(* Logix 5000 project; controller Savage_Saw vendor 1 type 14 code 154 rev 37.11; software revision 37.01 *)

TASK MainTask (continuous, watchdog 500 ms) : Init, Inputs, MainProgram, Outputs

MODULES
   Local : vendor 1 type 14 code 154 (PointIO 0, rev 37.11)
      RMC : vendor 590 type 43 code 5 (Ethernet 192.168.3.12, rev 1.1, StandardDataDriven RPI 20 ms, StandardDataDriven RPI 20 ms)
      RemoteHPU : 1734-AENTR (Ethernet 192.168.3.11, rev 7.13, Output RPI 20 ms)
         AnalogIn5_6 : 1734-IE2V (PointIO 1, rev 3.4, Input RPI 80 ms)
         InputDC0_8 : 1734-IB8 (PointIO 2, rev 3.22)
         InputDC9_15 : 1734-IB8 (PointIO 3, rev 3.22)
         OutputDC4_7 : vendor 1 type 7 code 134 (PointIO 5, rev 3.2)
         OutputDC0_3 : vendor 1 type 7 code 134 (PointIO 4, rev 3.2)
      Analog4_5 : 1734-IE2V (PointIO 4, rev 3.1, Input RPI 80 ms)
      Analog0_1 : 1734-IE2V (PointIO 2, rev 3.5, Input RPI 80 ms)
      Analog2_3 : 1734-IE2V (PointIO 3, rev 3.4, Input RPI 80 ms)
      Discrete_IO : Embedded (PointIO 1, rev 37.11, Output RPI 20 ms)
      SpindleSpeed : 1734-OE2V (PointIO 5, rev 3.5, Output RPI 50 ms)
      Swarf_Outputs : 1734-OA4 (PointIO 7, rev 3.22, Output RPI 20 ms)
      Light_Outputs : 1734-OA4 (PointIO 8, rev 3.22, Output RPI 20 ms)
      HPU_Outputs : 1734-OA4 (PointIO 6, rev 3.22, Output RPI 20 ms)
END_MODULES

TYPE AxisData :
STRUCT
   PositionActual : REAL;
   FinalOutput : REAL;
   VelocityActual : REAL;
   PositionTarget : REAL;
   VelocityTarget : REAL;
   InPosition : BOOL;
   AtVelocity : BOOL;
   OpenLoop : BOOL;
   FaultInput : BOOL;
   LimitPos : BOOL;
   LimitNeg : BOOL;
   Stopped : BOOL;
   InputEstimated : BOOL;
   OutputEnabled : BOOL;
   TargetGeneratorDone : BOOL;
   TargetGeneratorStateA : BOOL;
   TargetGeneratorStateB : BOOL;
   DirectOutput : BOOL;
   Enabled : BOOL;
   ExternalHalt : BOOL;
   Halted : BOOL;
   ForceControlled : BOOL;
   ForceLimitEnabled : BOOL;
   ForceLimited : BOOL;
   AtForce : BOOL;
   ForceInputEstimated : BOOL;
   ForceTargetGeneratorDone : BOOL;
   ForceTargetGeneratorStateA : BOOL;
   ForceTargetGeneratorStateB : BOOL;
   TargetGeneratorBusy : BOOL;
   ForceTargetGeneratorBusy : BOOL;
   FeedbackOK : BOOL;
   FeedbackOkSecondary : BOOL;
   StateMachineEnabled : BOOL;
   zs29 : BOOL;
   zs30 : BOOL;
   CommandAcknowledged : BOOL;
   Encoder_A_In : BOOL;
   Encoder_A_WireBreak : BOOL;
   Encoder_A_Fault : BOOL;
   Encoder_B_In : BOOL;
   Encoder_B_WireBreak : BOOL;
   Encoder_B_Fault : BOOL;
   Encoder_Z_In : BOOL;
   Encoder_Z_WireBreak : BOOL;
   Encoder_Z_Fault : BOOL;
   Encoder_Z_Learning : BOOL;
   HomeIn : BOOL;
   HomeFault : BOOL;
   HomeArmed : BOOL;
   HomeLatched : BOOL;
   RegistrationIn : BOOL;
   Registration0_Armed : BOOL;
   Registration0_Latched : BOOL;
   Registration1_Armed : BOOL;
   Registration1_Latched : BOOL;
   CommandMove : BOOL;
   CommandJog : BOOL;
   CommandStop : BOOL;
   CommandHome : BOOL;
   CommandZero : BOOL;
   CommandMoveRelative : BOOL;
   CommandClearZero : BOOL;
   z07 : BOOL;
   z08 : BOOL;
   z09 : BOOL;
   z10 : BOOL;
   z11 : BOOL;
   z12 : BOOL;
   z13 : BOOL;
   z14 : BOOL;
   z15 : BOOL;
   z16 : BOOL;
   z17 : BOOL;
   z18 : BOOL;
   z19 : BOOL;
   z20 : BOOL;
   z21 : BOOL;
   z22 : BOOL;
   z23 : BOOL;
   z24 : BOOL;
   z25 : BOOL;
   z26 : BOOL;
   z27 : BOOL;
   z28 : BOOL;
   z29 : BOOL;
   z30 : BOOL;
   z31 : BOOL;
   PositionDisplay : REAL;
   MoveComplete : BOOL;
   FollowingError : BOOL;
   ServoFault : BOOL;
   CommandAny : BOOL;
END_STRUCT
END_TYPE

TYPE Pass :
STRUCT
   WetPass : BOOL;
   Measure : BOOL;
   FeedRate : REAL;
   Depth : REAL;
   RemainDepth : REAL;
   EstimatedDiameter : REAL;
   MeasuredDiameter : REAL;
   FeedRateActual : REAL;
END_STRUCT
END_TYPE

VAR_GLOBAL   (* controller tags *)
   Auto : BOOL;
   AutoCutCancel : BOOL;
   AutoCutCancelFall : BOOL;
   AutoCutCancelOSF : BOOL;
   AutoCutReq : BOOL;
   AutoCutStartONS : BOOL;
   AutoCutStateChange : BOOL;
   AutoSpinCCW : BOOL;
   AutoSpinCW : BOOL;
   Axis : AxisData[3] := ([0].LimitPos := 1, [0].LimitNeg := 1, [0].OutputEnabled := 1, [0].TargetGeneratorDone := 1, [0].DirectOutput := 1, [0].Enabled := 1, [0].ForceControlled := 1, [0].ForceLimitEnabled := 1, [0].AtForce := 1, [0].ForceTargetGeneratorStateB := 1, [0].ForceTargetGeneratorBusy := 1, [0].zs30 := 1, [1].PositionActual := 1.5054715e-36, [1].OpenLoop := 1, [1].FaultInput := 1, [1].InputEstimated := 1, [1].TargetGeneratorStateA := 1, [1].TargetGeneratorStateB := 1, [1].Enabled := 1, [1].ExternalHalt := 1, [1].ForceControlled := 1, [1].ForceLimitEnabled := 1, [1].ForceLimited := 1, [1].ForceInputEstimated := 1, [1].ForceTargetGeneratorBusy := 1, [1].zs30 := 1, [2].PositionActual := 1.5054715e-36, [2].CommandAcknowledged := 1);
   AxisX_Gauge : ALIAS FOR Axis[0];
   AxisY_Traverse : ALIAS FOR Axis[1];
   AxisZ_RaiseLower : ALIAS FOR Axis[2];
   BladeChange10 : BOOL;
   BladeChange10ONS : BOOL;
   BladeChange20 : BOOL;
   BladeChange20ONS : BOOL;
   BladeChangeDone : BOOL;
   BladeChangeStartONS : BOOL;
   BladeChangeStateChange : BOOL;
   BladeMeasure10ONS : BOOL;
   BladeMeasure10StopAll : BOOL;
   BladeMeasure15ClearZero : BOOL;
   BladeMeasure20ONS : BOOL;
   BladeMeasure20Retract : BOOL;
   BladeMeasure30ONS : BOOL;
   BladeMeasure30Traverse : BOOL;
   BladeMeasure40Lower : BOOL;
   BladeMeasure40ONS : BOOL;
   BladeMeasure50ONS : BOOL;
   BladeMeasure50Stop : BOOL;
   BladeMeasure55ONS : BOOL;
   BladeMeasure55Raise : BOOL;
   BladeMeasure60ONS : BOOL;
   BladeMeasure60Stop : BOOL;
   BladeMeasure65Measure : BOOL;
   BladeMeasure65ONS : BOOL;
   BladeMeasure70Calc : BOOL;
   BladeMeasure70ONS : BOOL;
   BladeMeasure75ONS : BOOL;
   BladeMeasure75PartRef : BOOL;
   BladeMeasure80ONS : BOOL;
   BladeMeasure80Return : BOOL;
   BladeMeasureStartONS : BOOL;
   BladeMeasureStateChange : BOOL;
   BladeRadius : REAL;
   BladeRadiusKnown : BOOL;
   BuildCount : DINT;
   BuildDone : BOOL;
   BumpDistance : REAL;
   BumpDistanceDry : REAL;
   BumpDistanceWet : REAL;
   ClampPressure : REAL;
   CutEndPosition : REAL;
   CutForward : BOOL;
   CutOnReturn : BOOL;
   CutStartPosition : REAL;
   DryCutDepth : REAL;
   DryCutSpeed : REAL;
   DryPasses : DINT;
   Fault : BOOL;
   FaultOSR : BOOL;
   FaultRise : BOOL;
   GaugePotScale : REAL;
   GaugeVelocityHome : REAL;
   GaugeVelocityJogMax : REAL;
   GaugeVelocityMax : REAL;
   hmiFaultMessageNumber : DINT;
   HorsepowerActual : REAL;
   HorsepowerScale : REAL;
   HorsepowerTarget : REAL;
   HPUReadyToRun : BOOL;
   HydReady : BOOL;
   HydRun : BOOL;
   HydRunning : BOOL;
   HydStart : BOOL;
   HydStop : BOOL;
   inAnClampPressure : ALIAS FOR RemoteHPU:1:I.Ch0Data;
   InAnPotGauge : ALIAS FOR Local:3:I.Ch1Data;
   inAnPotRaiseLower : ALIAS FOR Local:2:I.Ch1Data;
   inAnPotTraverse : ALIAS FOR Local:3:I.Ch0Data;
   inAnServoPressure : ALIAS FOR RemoteHPU:1:I.Ch1Data;
   inAnSpindleSideA : ALIAS FOR Local:4:I.Ch0Data;
   inAnSpindlesideB : ALIAS FOR Local:4:I.Ch1Data;
   inAnSpindleSpeed : ALIAS FOR Local:2:I.Ch0Data;
   inFl01OilLevelWarning : ALIAS FOR RemoteHPU:3:I.0;
   inFl02OilLevelShutdownAlarm : ALIAS FOR RemoteHPU:3:I.2;
   inLs01OvertravelMnsGauge : ALIAS FOR Local:1:I.Data.8;
   inLs02OvertravelPlsGauge : ALIAS FOR Local:1:I.Data.9;
   inLs03OvertravelMnsTraverse : ALIAS FOR Local:1:I.Data.10;
   inLs04OvertravelPlsTraverse : ALIAS FOR Local:1:I.Data.11;
   inLs05OvertravelMnsRaiseLower : ALIAS FOR Local:1:I.Data.12;
   inLs06OvertravelPlsRaiseLower : ALIAS FOR Local:1:I.Data.13;
   inLs07BladeGuard : ALIAS FOR Local:1:I.Data.14;
   inMS1HydraulicPump : ALIAS FOR Local:1:I.Data.1;
   inMS2HydraulicLoopPump : ALIAS FOR Local:1:I.Data.2;
   inMS3HydCoolingFan : ALIAS FOR Local:1:I.Data.3;
   inMS4CoolantPump : ALIAS FOR Local:1:I.Data.4;
   inMS5SwarfPump : ALIAS FOR Local:1:I.Data.5;
   inMS6SwarfConveyor : ALIAS FOR Local:1:I.Data.6;
   inPe01BladeDetect : ALIAS FOR Local:1:I.Data.7;
   inPs01LoopFilterDirty : ALIAS FOR RemoteHPU:2:I.5;
   inPs02PressureFilterDirty : ALIAS FOR RemoteHPU:2:I.6;
   inPs03MotorCaseDrain : ALIAS FOR RemoteHPU:2:I.7;
   inPs04SwarfFilterDirty : ALIAS FOR Local:1:I.Data.15;
   inPx01Pump1Inlet : ALIAS FOR RemoteHPU:2:I.0;
   inPx02Pump2Inlet : ALIAS FOR RemoteHPU:2:I.1;
   InPx03PumpAA4Inlet : ALIAS FOR RemoteHPU:2:I.2;
   inPx04LoopInlet : ALIAS FOR RemoteHPU:2:I.3;
   inPx05DrainValve : ALIAS FOR RemoteHPU:2:I.4;
   inSpare746 : ALIAS FOR RemoteHPU:3:I.4;
   inSpare747 : ALIAS FOR RemoteHPU:3:I.5;
   inSR1SafetyRelay : ALIAS FOR Local:1:I.Data.0;
   inTs01OilTempWarning : ALIAS FOR RemoteHPU:3:I.1;
   inTs02OilTempShutdownAlarm : ALIAS FOR RemoteHPU:3:I.3;
   LastCutDepth : REAL;
   LastCutSpeed : REAL;
   MC_Reset : ALIAS FOR RMC:O2.Data[3].0;
   NorthZero : BOOL;
   OilWarm : BOOL;
   outAnSpindleMotor : ALIAS FOR Local:5:O.Ch1Data;
   outAnSpindlePump : ALIAS FOR Local:5:O.Ch0Data;
   outCr01BrakeTraverse : ALIAS FOR RemoteHPU:4:O.0;
   outCr02BrakeGauge : ALIAS FOR RemoteHPU:4:O.1;
   outCr03BrakeRaiseLower : ALIAS FOR RemoteHPU:4:O.2;
   outCr04ClampAdvance : ALIAS FOR RemoteHPU:5:O.0;
   outCr05GageGripperAdvance : ALIAS FOR RemoteHPU:5:O.1;
   outCrlLaserLight : ALIAS FOR Local:8:O.Data.0;
   outLtaStackLtAmber : ALIAS FOR Local:8:O.Data.2;
   outLtgStackLtGreen : ALIAS FOR Local:8:O.Data.1;
   outLtrStackLtRed : ALIAS FOR Local:8:O.Data.3;
   outMs1HydrulicPump : ALIAS FOR Local:6:O.Data.0;
   outMs2LoopPump : ALIAS FOR Local:6:O.Data.1;
   outMs3HydraulicCoolFan : ALIAS FOR Local:6:O.Data.2;
   outMs4Coolant : ALIAS FOR Local:6:O.Data.3;
   outMs5SwarfPump : ALIAS FOR Local:7:O.Data.0;
   outMs6SwarfConveyor : ALIAS FOR Local:7:O.Data.1;
   outSpare632 : ALIAS FOR Local:7:O.Data.2;
   outSpare633 : ALIAS FOR Local:7:O.Data.3;
   outSpare806 : ALIAS FOR RemoteHPU:4:O.3;
   outSpare817 : ALIAS FOR RemoteHPU:5:O.2;
   outSpare818 : ALIAS FOR RemoteHPU:5:O.3;
   Pass : Pass[21];
   PastPart : REAL;
   Pi : REAL := 3.1415927; {constant}
   RaiseLowerPotScale : REAL;
   RaiseLowerVelocityHome : REAL;
   RaiseLowerVelocityJogMax : REAL;
   RaiseLowerVelocityMax : REAL;
   RemainDepth : REAL;
   RpmTarget : REAL;
   RpmTarget105Pct : REAL;
   SafetyRelayAutoReset : BOOL;
   ServoPressure : REAL;
   SFPM : REAL;
   SpinCCWActive : BOOL;
   SpinCCWDemand : BOOL;
   SpinCWActive : BOOL;
   SpinCWDemand : BOOL;
   SpinDemandFall : BOOL;
   SpindleMotorOutputScale : REAL;
   SpindlePressure : REAL;
   SpindlePressureCCW : REAL;
   SpindlePressureCW : REAL;
   SpindlePressureDisplay : REAL;
   SpindlePressureScale : REAL;
   SpindlePressureTarget : REAL;
   SpindleRPM : REAL;
   SpindleRPMAtTarget : BOOL;
   SpindleRPMError : REAL;
   SpindleRPMGate : REAL;
   SpindleStall : BOOL;
   SpindleStallPressure : REAL;
   SpindleStallRPM : REAL;
   State : DINT;
   State200Build : BOOL;
   State200ONS : BOOL;
   State205 : BOOL;
   State205ONS : BOOL;
   State207ONS : BOOL;
   State207TraverseInitial : BOOL;
   State210Direction : BOOL;
   State210ONS : BOOL;
   State220ONS : BOOL;
   State220TraverseToStart : BOOL;
   State230StartSaw : BOOL;
   State240 : BOOL;
   State240ONS : BOOL;
   State250CheckRPM : BOOL;
   State250ONS : BOOL;
   State260Cut : BOOL;
   State260ONS : BOOL;
   State280 : BOOL;
   State280ONS : BOOL;
   State285BladeMeasure : BOOL;
   State290ONS : BOOL;
   State290RaiseBlade : BOOL;
   State299 : BOOL;
   StepCount : DINT;
   tbA1JogIn : BOOL;
   tbA1JogOut : BOOL;
   tbA2JogMinus : BOOL;
   tbA2JogPlus : BOOL;
   tbA3JogMinus : BOOL;
   tbA3JogPlus : BOOL;
   tbAutoCut : BOOL;
   tbAutoCutONS : BOOL;
   tbAutoGauge : BOOL;
   tbAutoWet : BOOL;
   tbBladeChange : BOOL;
   tbBladeCompensation : BOOL;
   tbBladeMeasure : BOOL;
   tbCCW : BOOL;
   tbCoolant : BOOL;
   tbCW : BOOL;
   tbDryBump : BOOL;
   tbGaugeClamp : BOOL;
   tbGaugeUnclamp : BOOL;
   tbHome : BOOL;
   tbLaser : BOOL;
   tbMS1HydPump : BOOL;
   tbMS2LoopPump : BOOL;
   tbMS3HydCoolingFan : BOOL;
   tbMS4CoolantPump : BOOL;
   tbMS5SwarfPump : BOOL;
   tbMS6SwarfConveyor : BOOL;
   tbNorthRef : BOOL;
   tbOnOff : BOOL;
   tbPlateMeasure : BOOL;
   tbSouthRef : BOOL;
   tbWetBump : BOOL;
   tbWorkClamp : BOOL;
   tbWorkUnclamp : BOOL;
   tbZeroGauge : BOOL;
   Thickness : REAL;
   timerAxisZ_RaiseLowerClearZero : TIMER := (PRE := 1000);
   timerGaugeBrakeDelay : TIMER := (PRE := 2000);
   timerRaiseLowerBrakeDelay : TIMER := (PRE := 2000);
   timerSpindleStall : TIMER := (PRE := 3000);
   timerState250CheckRPM : TIMER;
   timerTraverseBrakeDelay : TIMER := (PRE := 2000);
   TraversePotScale : REAL;
   TraverseRange : REAL;
   TraverseVelocityHome : REAL;
   TraverseVelocityJogMax : REAL;
   TraverseVelocityMax : REAL;
   ValidData : BOOL;
   WetCutDepth : REAL;
   WetCutSpeed : REAL;
   WetPasses : DINT;
   Width : REAL;
   X_AutoCut : BOOL;
   X_BladeChange : BOOL;
   X_BladeMeasure : BOOL;
   X_Fault : BOOL;
   X_Homing : BOOL;
   X_Manual : BOOL;
   X_Off : BOOL;
   X_State : DINT;
END_VAR

PROGRAM Init   (* main routine Init *)
VAR
   Initialized : BOOL;
END_VAR

ROUTINE Init   (* ladder *)
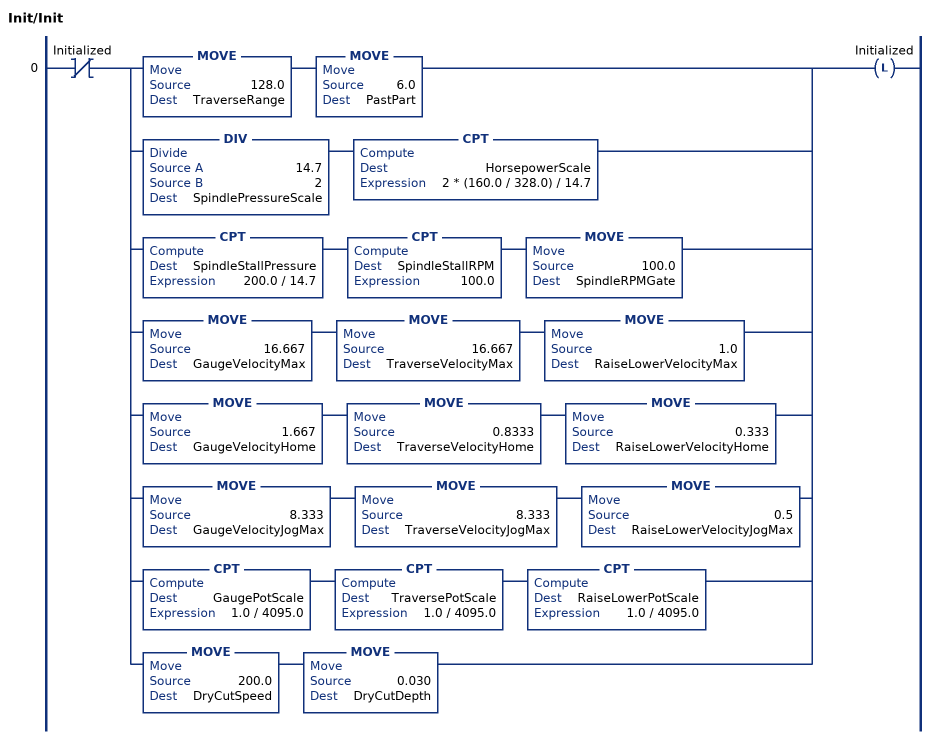
   0: XIO(Initialized)[MOVE(128.0,TraverseRange) MOVE(6.0,PastPart) ,DIV(14.7,2,SpindlePressureScale) CPT(HorsepowerScale,2 * (160.0 / 328.0) / 14.7) ,CPT(SpindleStallPressure,200.0 / 14.7) CPT(SpindleStallRPM,100.0) MOVE(100.0,SpindleRPMGate) ,MOVE(16.667,GaugeVelocityMax) MOVE(16.667,TraverseVelocityMax) MOVE(1.0,RaiseLowerVelocityMax) ,MOVE(1.667,GaugeVelocityHome) MOVE(0.8333,TraverseVelocityHome) MOVE(0.333,RaiseLowerVelocityHome) ,MOVE(8.333,GaugeVelocityJogMax) MOVE(8.333,TraverseVelocityJogMax) MOVE(0.5,RaiseLowerVelocityJogMax) ,CPT(GaugePotScale,1.0 / 4095.0) CPT(TraversePotScale,1.0 / 4095.0) CPT(RaiseLowerPotScale,1.0 / 4095.0) ,MOVE(200.0,DryCutSpeed) MOVE(0.030,DryCutDepth) ]OTL(Initialized);
END_ROUTINE
END_PROGRAM

PROGRAM Inputs   (* main routine Inputs *)
VAR
   iAxis : DINT;
END_VAR

ROUTINE Inputs   (* ladder *)
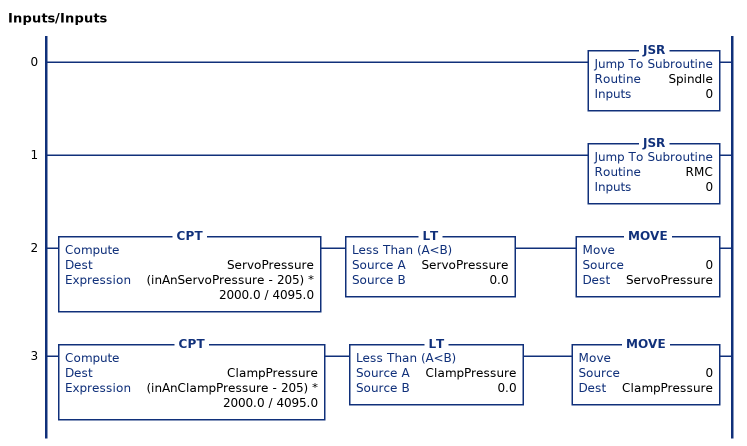
   0: JSR(Spindle,0);
   1: JSR(RMC,0);
   2: CPT(ServoPressure,(inAnServoPressure - 205) * 2000.0 / 4095.0)LT(ServoPressure,0.0)MOVE(0,ServoPressure);
   3: CPT(ClampPressure,(inAnClampPressure - 205) * 2000.0 / 4095.0)LT(ClampPressure,0.0)MOVE(0,ClampPressure);
END_ROUTINE

ROUTINE RMC   (* ladder *)
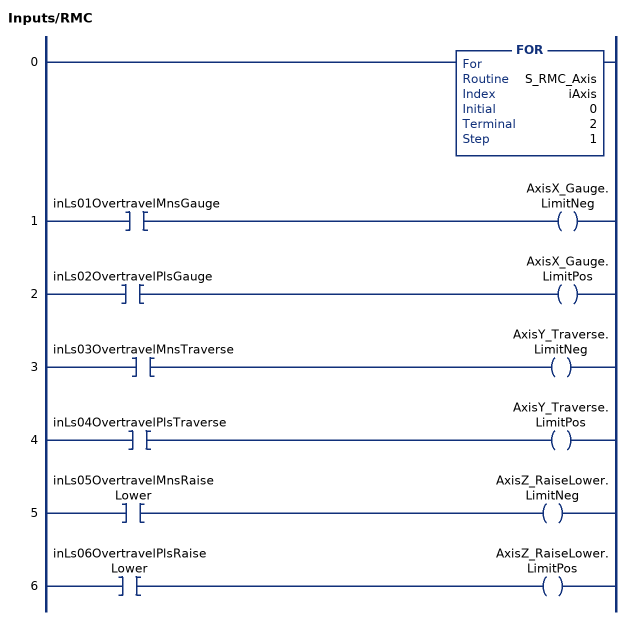
   0: FOR(S_RMC_Axis,iAxis,0,2,1);
   1: XIC(inLs01OvertravelMnsGauge)OTE(AxisX_Gauge.LimitNeg);
   2: XIC(inLs02OvertravelPlsGauge)OTE(AxisX_Gauge.LimitPos);
   3: XIC(inLs03OvertravelMnsTraverse)OTE(AxisY_Traverse.LimitNeg);
   4: XIC(inLs04OvertravelPlsTraverse)OTE(AxisY_Traverse.LimitPos);
   5: XIC(inLs05OvertravelMnsRaiseLower)OTE(AxisZ_RaiseLower.LimitNeg);
   6: XIC(inLs06OvertravelPlsRaiseLower)OTE(AxisZ_RaiseLower.LimitPos);
END_ROUTINE

ROUTINE S_RMC_Axis   (* ladder *)
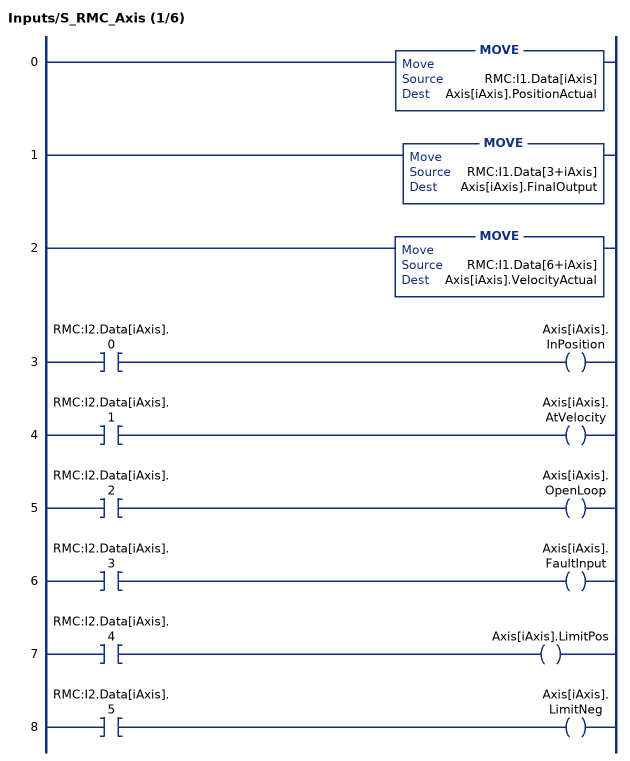
   0: MOVE(RMC:I1.Data[iAxis],Axis[iAxis].PositionActual);
   1: MOVE(RMC:I1.Data[3+iAxis],Axis[iAxis].FinalOutput);
   2: MOVE(RMC:I1.Data[6+iAxis],Axis[iAxis].VelocityActual);
   3: XIC(RMC:I2.Data[iAxis].0)OTE(Axis[iAxis].InPosition);
   4: XIC(RMC:I2.Data[iAxis].1)OTE(Axis[iAxis].AtVelocity);
   5: XIC(RMC:I2.Data[iAxis].2)OTE(Axis[iAxis].OpenLoop);
   6: XIC(RMC:I2.Data[iAxis].3)OTE(Axis[iAxis].FaultInput);
   7: XIC(RMC:I2.Data[iAxis].4)OTE(Axis[iAxis].LimitPos);
   8: XIC(RMC:I2.Data[iAxis].5)OTE(Axis[iAxis].LimitNeg);
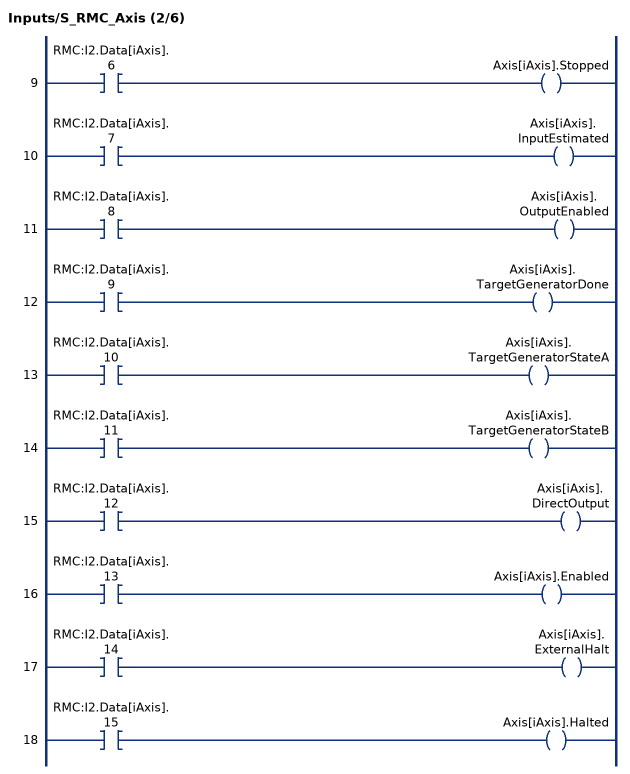
   9: XIC(RMC:I2.Data[iAxis].6)OTE(Axis[iAxis].Stopped);
   10: XIC(RMC:I2.Data[iAxis].7)OTE(Axis[iAxis].InputEstimated);
   11: XIC(RMC:I2.Data[iAxis].8)OTE(Axis[iAxis].OutputEnabled);
   12: XIC(RMC:I2.Data[iAxis].9)OTE(Axis[iAxis].TargetGeneratorDone);
   13: XIC(RMC:I2.Data[iAxis].10)OTE(Axis[iAxis].TargetGeneratorStateA);
   14: XIC(RMC:I2.Data[iAxis].11)OTE(Axis[iAxis].TargetGeneratorStateB);
   15: XIC(RMC:I2.Data[iAxis].12)OTE(Axis[iAxis].DirectOutput);
   16: XIC(RMC:I2.Data[iAxis].13)OTE(Axis[iAxis].Enabled);
   17: XIC(RMC:I2.Data[iAxis].14)OTE(Axis[iAxis].ExternalHalt);
   18: XIC(RMC:I2.Data[iAxis].15)OTE(Axis[iAxis].Halted);
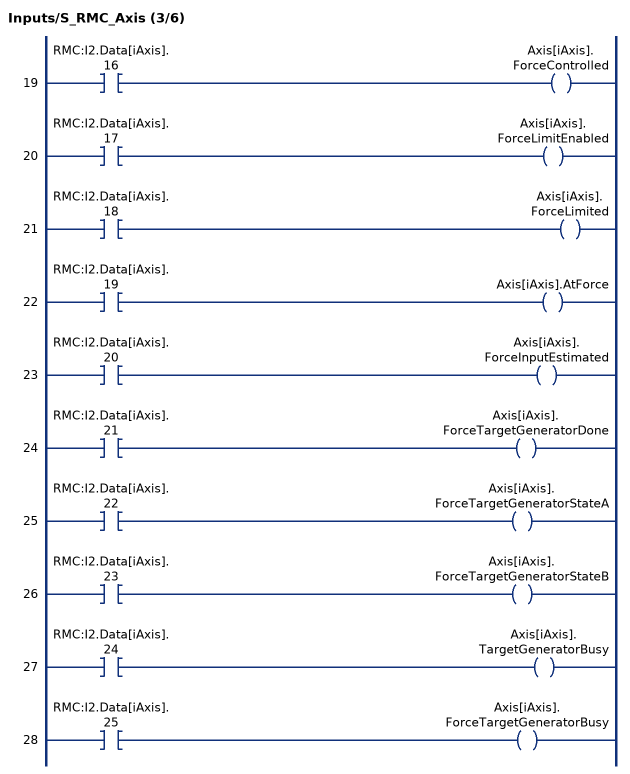
   19: XIC(RMC:I2.Data[iAxis].16)OTE(Axis[iAxis].ForceControlled);
   20: XIC(RMC:I2.Data[iAxis].17)OTE(Axis[iAxis].ForceLimitEnabled);
   21: XIC(RMC:I2.Data[iAxis].18)OTE(Axis[iAxis].ForceLimited);
   22: XIC(RMC:I2.Data[iAxis].19)OTE(Axis[iAxis].AtForce);
   23: XIC(RMC:I2.Data[iAxis].20)OTE(Axis[iAxis].ForceInputEstimated);
   24: XIC(RMC:I2.Data[iAxis].21)OTE(Axis[iAxis].ForceTargetGeneratorDone);
   25: XIC(RMC:I2.Data[iAxis].22)OTE(Axis[iAxis].ForceTargetGeneratorStateA);
   26: XIC(RMC:I2.Data[iAxis].23)OTE(Axis[iAxis].ForceTargetGeneratorStateB);
   27: XIC(RMC:I2.Data[iAxis].24)OTE(Axis[iAxis].TargetGeneratorBusy);
   28: XIC(RMC:I2.Data[iAxis].25)OTE(Axis[iAxis].ForceTargetGeneratorBusy);
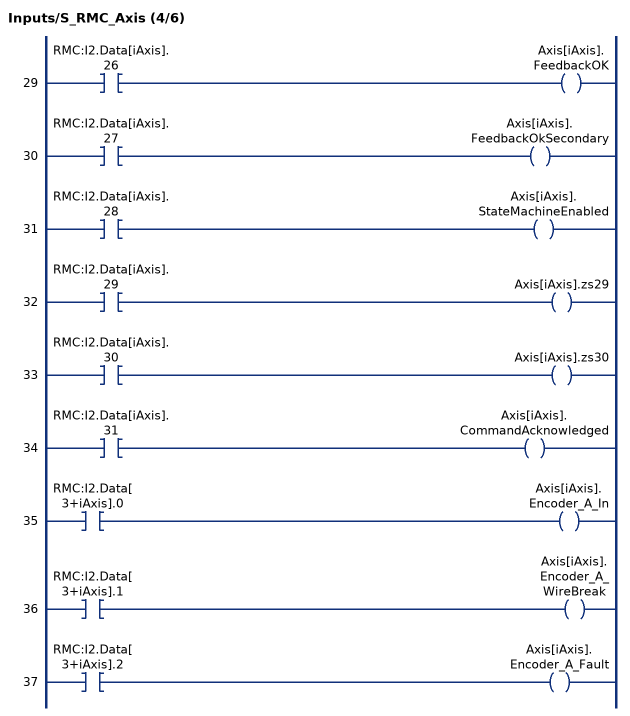
   29: XIC(RMC:I2.Data[iAxis].26)OTE(Axis[iAxis].FeedbackOK);
   30: XIC(RMC:I2.Data[iAxis].27)OTE(Axis[iAxis].FeedbackOkSecondary);
   31: XIC(RMC:I2.Data[iAxis].28)OTE(Axis[iAxis].StateMachineEnabled);
   32: XIC(RMC:I2.Data[iAxis].29)OTE(Axis[iAxis].zs29);
   33: XIC(RMC:I2.Data[iAxis].30)OTE(Axis[iAxis].zs30);
   34: XIC(RMC:I2.Data[iAxis].31)OTE(Axis[iAxis].CommandAcknowledged);
   35: XIC(RMC:I2.Data[3+iAxis].0)OTE(Axis[iAxis].Encoder_A_In);
   36: XIC(RMC:I2.Data[3+iAxis].1)OTE(Axis[iAxis].Encoder_A_WireBreak);
   37: XIC(RMC:I2.Data[3+iAxis].2)OTE(Axis[iAxis].Encoder_A_Fault);
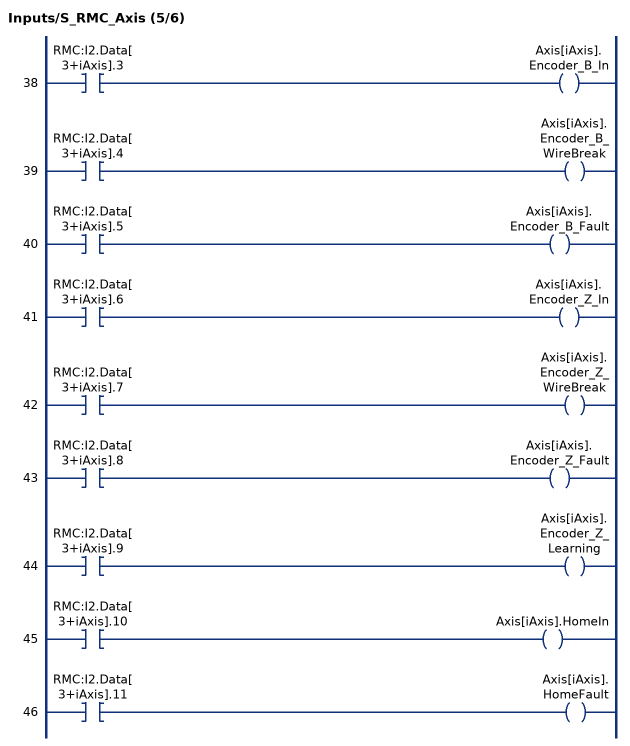
   38: XIC(RMC:I2.Data[3+iAxis].3)OTE(Axis[iAxis].Encoder_B_In);
   39: XIC(RMC:I2.Data[3+iAxis].4)OTE(Axis[iAxis].Encoder_B_WireBreak);
   40: XIC(RMC:I2.Data[3+iAxis].5)OTE(Axis[iAxis].Encoder_B_Fault);
   41: XIC(RMC:I2.Data[3+iAxis].6)OTE(Axis[iAxis].Encoder_Z_In);
   42: XIC(RMC:I2.Data[3+iAxis].7)OTE(Axis[iAxis].Encoder_Z_WireBreak);
   43: XIC(RMC:I2.Data[3+iAxis].8)OTE(Axis[iAxis].Encoder_Z_Fault);
   44: XIC(RMC:I2.Data[3+iAxis].9)OTE(Axis[iAxis].Encoder_Z_Learning);
   45: XIC(RMC:I2.Data[3+iAxis].10)OTE(Axis[iAxis].HomeIn);
   46: XIC(RMC:I2.Data[3+iAxis].11)OTE(Axis[iAxis].HomeFault);
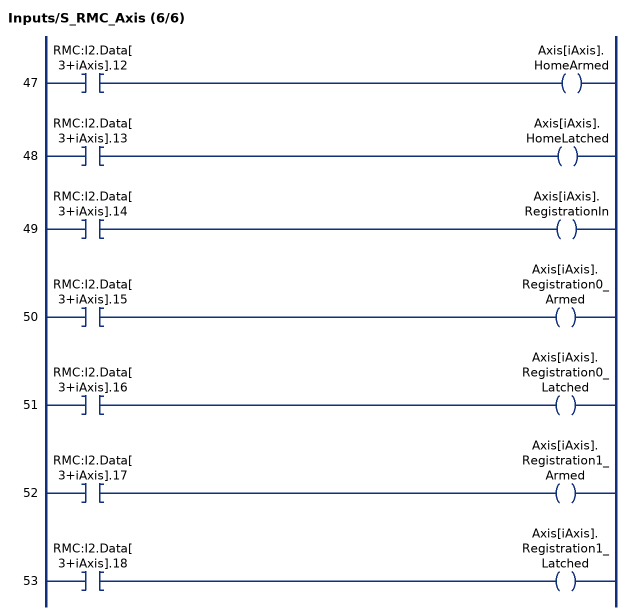
   47: XIC(RMC:I2.Data[3+iAxis].12)OTE(Axis[iAxis].HomeArmed);
   48: XIC(RMC:I2.Data[3+iAxis].13)OTE(Axis[iAxis].HomeLatched);
   49: XIC(RMC:I2.Data[3+iAxis].14)OTE(Axis[iAxis].RegistrationIn);
   50: XIC(RMC:I2.Data[3+iAxis].15)OTE(Axis[iAxis].Registration0_Armed);
   51: XIC(RMC:I2.Data[3+iAxis].16)OTE(Axis[iAxis].Registration0_Latched);
   52: XIC(RMC:I2.Data[3+iAxis].17)OTE(Axis[iAxis].Registration1_Armed);
   53: XIC(RMC:I2.Data[3+iAxis].18)OTE(Axis[iAxis].Registration1_Latched);
END_ROUTINE

ROUTINE Spindle   (* ladder *)
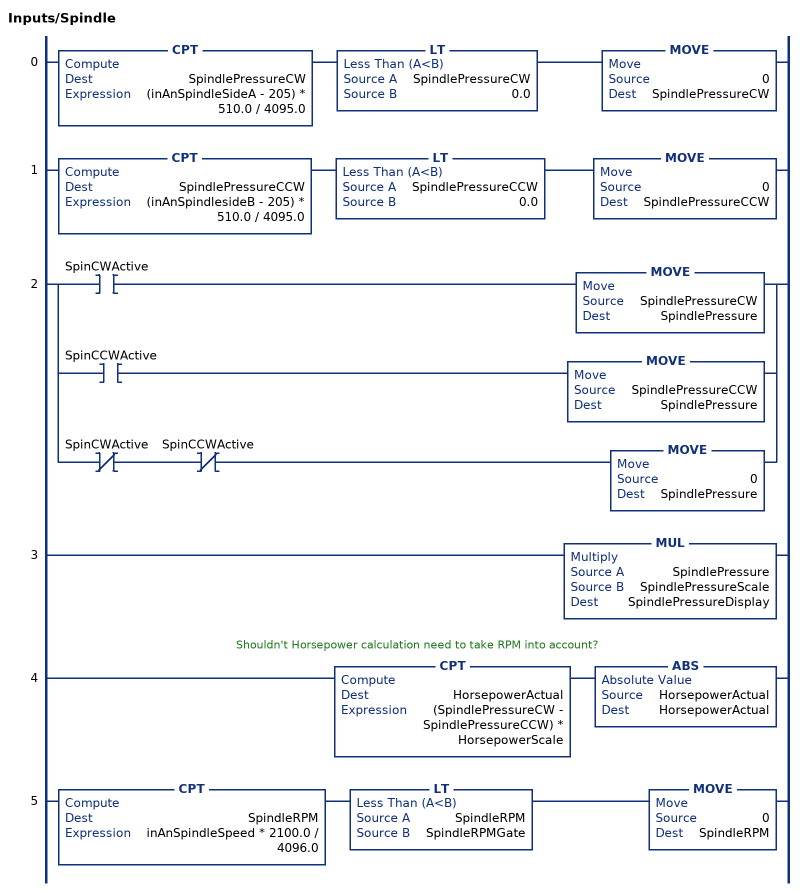
   0: CPT(SpindlePressureCW,(inAnSpindleSideA - 205) * 510.0 / 4095.0)LT(SpindlePressureCW,0.0)MOVE(0,SpindlePressureCW);
   1: CPT(SpindlePressureCCW,(inAnSpindlesideB - 205) * 510.0 / 4095.0)LT(SpindlePressureCCW,0.0)MOVE(0,SpindlePressureCCW);
   2: [XIC(SpinCWActive) MOVE(SpindlePressureCW,SpindlePressure) ,XIC(SpinCCWActive) MOVE(SpindlePressureCCW,SpindlePressure) ,XIO(SpinCWActive) XIO(SpinCCWActive) MOVE(0,SpindlePressure) ];
   3: MUL(SpindlePressure,SpindlePressureScale,SpindlePressureDisplay);
   // Shouldn't Horsepower calculation need to take RPM into account?
   4: CPT(HorsepowerActual,(SpindlePressureCW - SpindlePressureCCW) * HorsepowerScale)ABS(HorsepowerActual,HorsepowerActual);
   5: CPT(SpindleRPM,inAnSpindleSpeed * 2100.0 / 4096.0)LT(SpindleRPM,SpindleRPMGate)MOVE(0,SpindleRPM);
END_ROUTINE
END_PROGRAM

PROGRAM MainProgram   (* main routine Main *)
VAR
   AnyJogRise : BOOL;
   AnyJogStorage : BOOL;
   btHpuValvesOK : BOOL;
   HydRunFall : BOOL;
   HydRunFallStorage : BOOL;
   HydRunRise : BOOL;
   HydRunRiseStorage : BOOL;
   iAxis : DINT := 2;
   ManualSpinCCW : BOOL;
   ManualSpinCW : BOOL;
   SafetyRelayAutoResetDelayStorage : BOOL;
   spinActive : BOOL;
   spinDemand : BOOL;
   tbHydSShot : BOOL;
   tbHydSShotStorage : BOOL;
   timerSafetyRelayDelay : TIMER := (PRE := 1000);
   timerSpinDownCCW : TIMER := (PRE := 2000);
   timerSpinDownCW : TIMER := (PRE := 2000);
   tmrHydLoopDelay : TIMER := (PRE := 2000);
END_VAR

ROUTINE Calc   (* structured text *)
   if BladeRadius > 1 then
   	RpmTarget := (SFPM / Pi) * 120.00 / (2 * BladeRadius);
   else
   	RpmTarget := 0.0;
   end_if;
   
   SpindlePressureTarget := (HorsepowerTarget * 328.0 / 160.0 + 22.0) * 14.7;
   if SpindlePressureTarget > 350.0 * 14.7 then
   	SpindlePressureTarget := 350.0 * 14.7;
   end_if;
   
   if State200Build then
   	BuildCount := 0;
   	RemainDepth := Thickness;
   
   	if WetPasses > 1 then
   		WetCutDepth := 0.00001 + (Thickness - (DryPasses * DryCutDepth) - LastCutDepth) / (WetPasses - 1);
   	else
   		WetCutDepth := 0;
   	end_if;
   
   	while BuildCount <= 20 do
   		Pass[BuildCount].WetPass := 1;
   		if DryPasses > BuildCount then
   			Pass[BuildCount].WetPass := 0;
   			Pass[BuildCount].FeedRate := DryCutSpeed;
   			Pass[BuildCount].Depth := DryCutDepth;
   		elsif (WetPasses - 1) + DryPasses > BuildCount then
   			Pass[BuildCount].FeedRate := WetCutSpeed;
   			Pass[BuildCount].Depth := WetCutDepth;
   		elsif (WetPasses - 1) + DryPasses = BuildCount then
   			Pass[BuildCount].FeedRate := LastCutSpeed;
   			Pass[BuildCount].Depth := LastCutDepth;
   		end_if;
   		RemainDepth := RemainDepth - Pass[BuildCount].Depth;
   		Pass[BuildCount].RemainDepth := RemainDepth;
   		BuildCount := BuildCount + 1;
   	end_while;
   
   	BuildDone := 1;
   end_if;
END_ROUTINE

ROUTINE Conditions   (* ladder *)
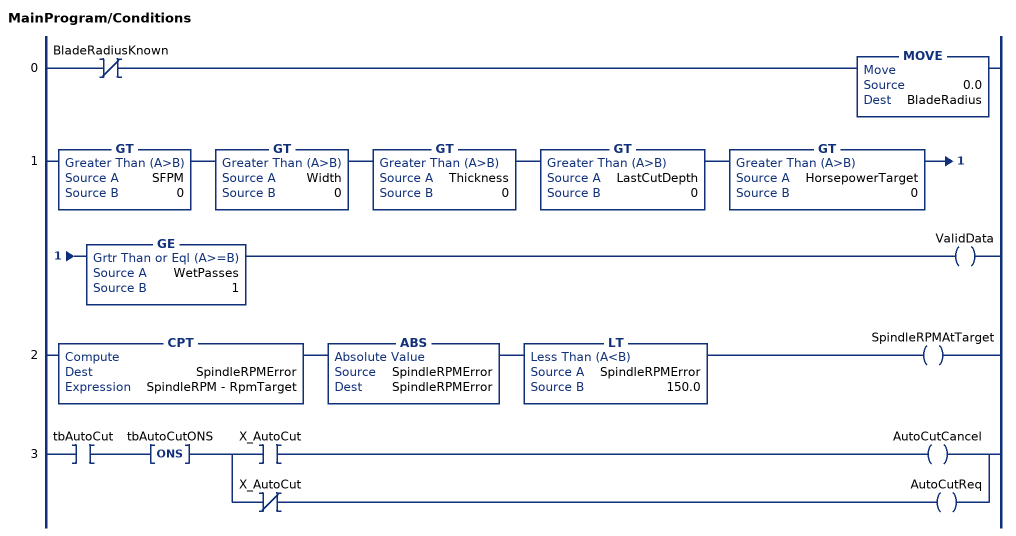
   0: XIO(BladeRadiusKnown)MOVE(0.0,BladeRadius);
   1: GT(SFPM,0)GT(Width,0)GT(Thickness,0)GT(LastCutDepth,0)GT(HorsepowerTarget,0)GE(WetPasses,1)OTE(ValidData);
   2: CPT(SpindleRPMError,SpindleRPM - RpmTarget)ABS(SpindleRPMError,SpindleRPMError)LT(SpindleRPMError,150.0)OTE(SpindleRPMAtTarget);
   3: XIC(tbAutoCut)ONS(tbAutoCutONS)[XIC(X_AutoCut) OTE(AutoCutCancel) ,XIO(X_AutoCut) OTE(AutoCutReq) ];
END_ROUTINE

ROUTINE Main   (* ladder *)
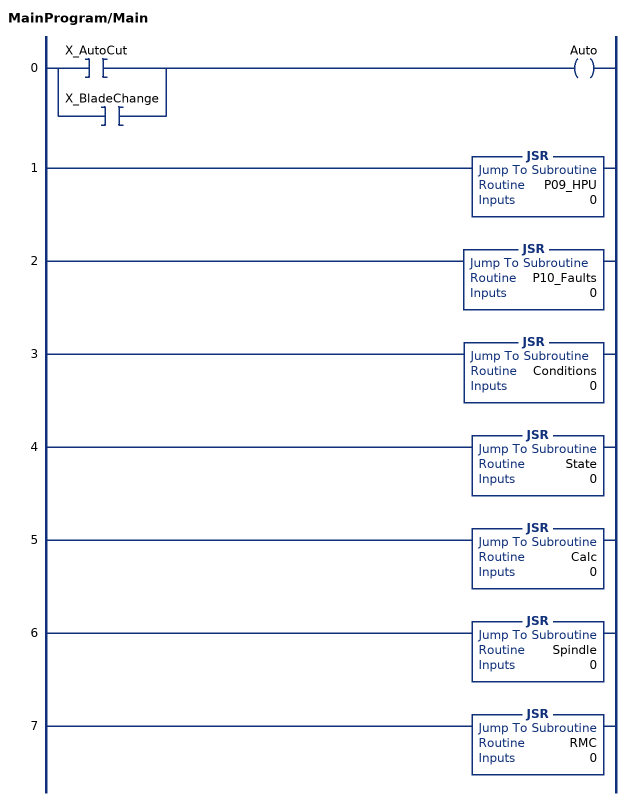
   0: [XIC(X_AutoCut) ,XIC(X_BladeChange) ]OTE(Auto);
   1: JSR(P09_HPU,0);
   2: JSR(P10_Faults,0);
   3: JSR(Conditions,0);
   4: JSR(State,0);
   5: JSR(Calc,0);
   6: JSR(Spindle,0);
   7: JSR(RMC,0);
END_ROUTINE

ROUTINE P09_HPU   (* ladder *)
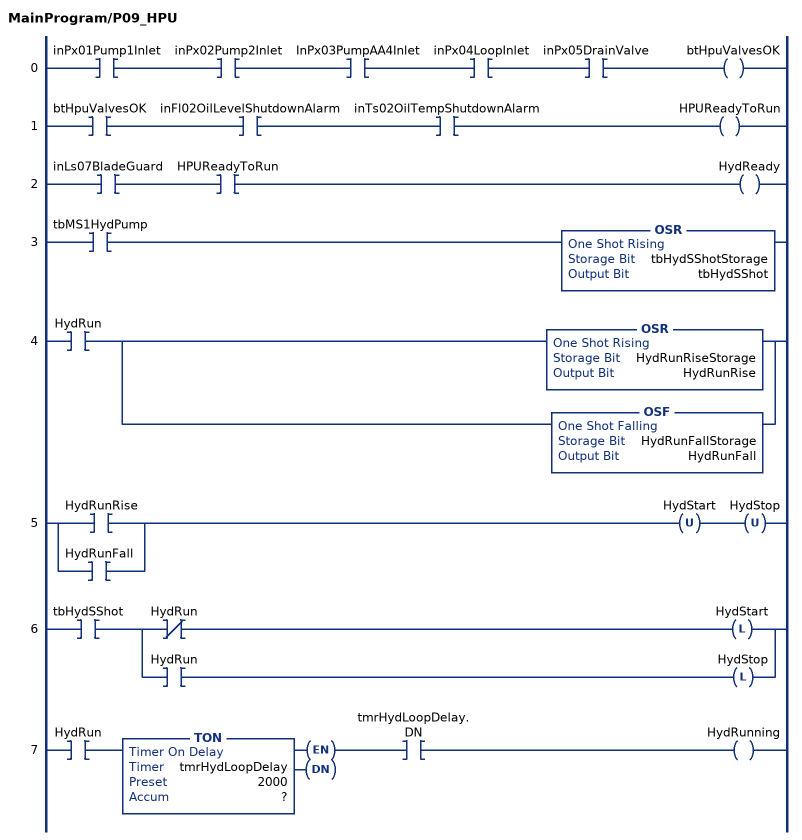
   0: XIC(inPx01Pump1Inlet)XIC(inPx02Pump2Inlet)XIC(InPx03PumpAA4Inlet)XIC(inPx04LoopInlet)XIC(inPx05DrainValve)OTE(btHpuValvesOK);
   1: XIC(btHpuValvesOK)XIC(inFl02OilLevelShutdownAlarm)XIC(inTs02OilTempShutdownAlarm)OTE(HPUReadyToRun);
   2: XIC(inLs07BladeGuard)XIC(HPUReadyToRun)OTE(HydReady);
   3: XIC(tbMS1HydPump)OSR(tbHydSShotStorage,tbHydSShot);
   4: XIC(HydRun)[OSR(HydRunRiseStorage,HydRunRise) ,OSF(HydRunFallStorage,HydRunFall) ];
   5: [XIC(HydRunRise) ,XIC(HydRunFall) ]OTU(HydStart)OTU(HydStop);
   6: XIC(tbHydSShot)[XIO(HydRun) OTL(HydStart) ,XIC(HydRun) OTL(HydStop) ];
   7: XIC(HydRun)TON(tmrHydLoopDelay,?,?)XIC(tmrHydLoopDelay.DN)OTE(HydRunning);
END_ROUTINE

ROUTINE P10_Faults   (* ladder *)
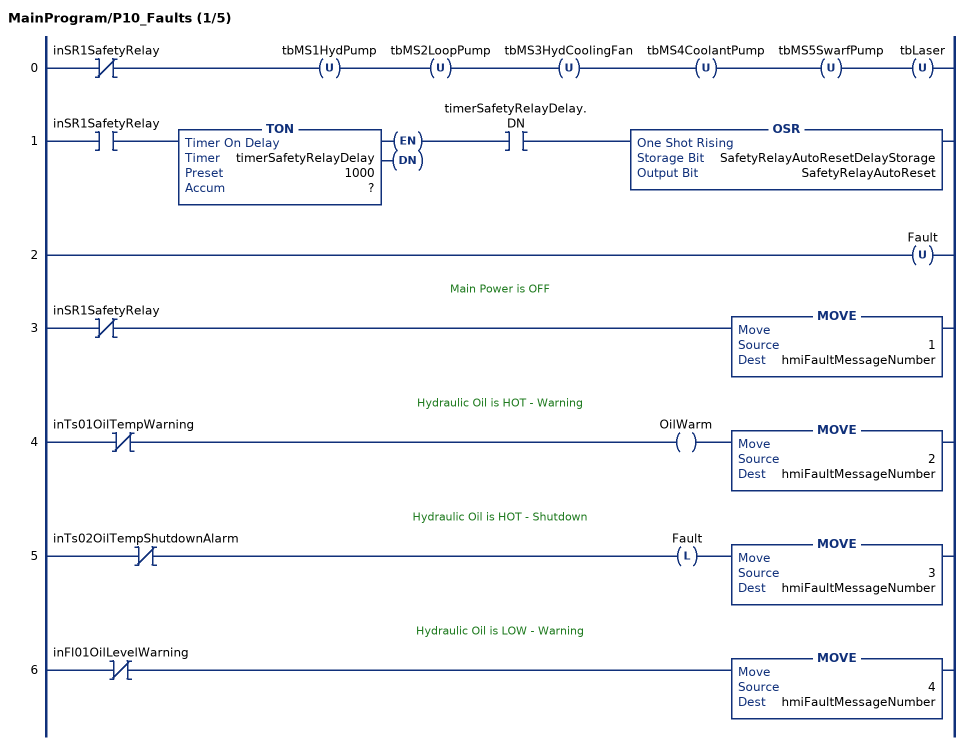
   0: XIO(inSR1SafetyRelay)OTU(tbMS1HydPump)OTU(tbMS2LoopPump)OTU(tbMS3HydCoolingFan)OTU(tbMS4CoolantPump)OTU(tbMS5SwarfPump)OTU(tbLaser);
   1: XIC(inSR1SafetyRelay)TON(timerSafetyRelayDelay,?,?)XIC(timerSafetyRelayDelay.DN)OSR(SafetyRelayAutoResetDelayStorage,SafetyRelayAutoReset);
   2: OTU(Fault);
   // Main Power is OFF
   3: XIO(inSR1SafetyRelay)MOVE(1,hmiFaultMessageNumber);
   // Hydraulic Oil is HOT - Warning
   4: XIO(inTs01OilTempWarning)OTE(OilWarm)MOVE(2,hmiFaultMessageNumber);
   // Hydraulic Oil is HOT - Shutdown
   5: XIO(inTs02OilTempShutdownAlarm)OTL(Fault)MOVE(3,hmiFaultMessageNumber);
   // Hydraulic Oil is LOW - Warning
   6: XIO(inFl01OilLevelWarning)MOVE(4,hmiFaultMessageNumber);
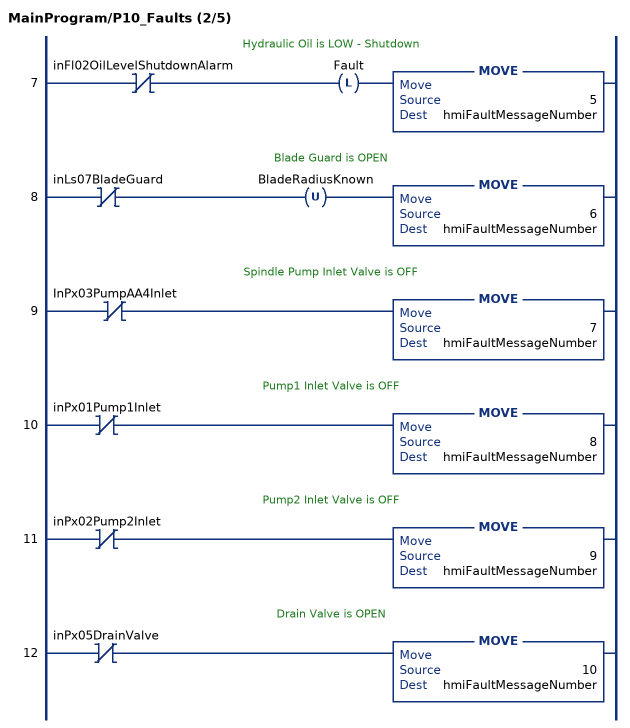
   // Hydraulic Oil is LOW - Shutdown
   7: XIO(inFl02OilLevelShutdownAlarm)OTL(Fault)MOVE(5,hmiFaultMessageNumber);
   // Blade Guard is OPEN
   8: XIO(inLs07BladeGuard)OTU(BladeRadiusKnown)MOVE(6,hmiFaultMessageNumber);
   // Spindle Pump Inlet Valve is OFF
   9: XIO(InPx03PumpAA4Inlet)MOVE(7,hmiFaultMessageNumber);
   // Pump1 Inlet Valve is OFF
   10: XIO(inPx01Pump1Inlet)MOVE(8,hmiFaultMessageNumber);
   // Pump2 Inlet Valve is OFF
   11: XIO(inPx02Pump2Inlet)MOVE(9,hmiFaultMessageNumber);
   // Drain Valve is OPEN
   12: XIO(inPx05DrainValve)MOVE(10,hmiFaultMessageNumber);
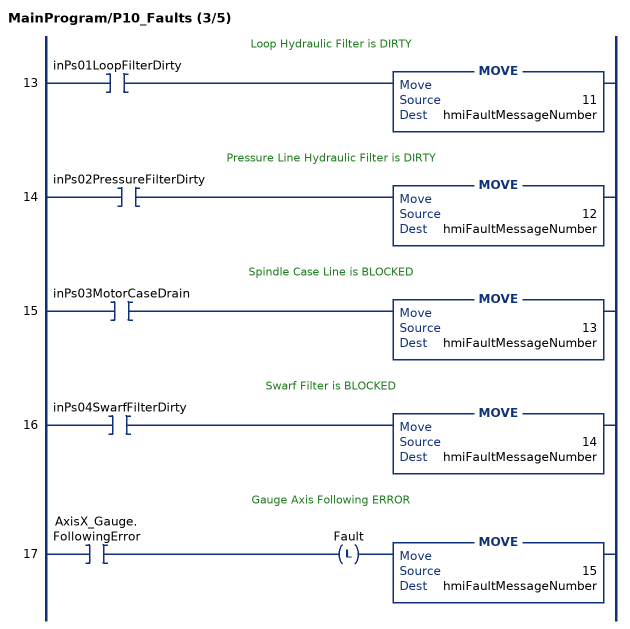
   // Loop Hydraulic Filter is DIRTY
   13: XIC(inPs01LoopFilterDirty)MOVE(11,hmiFaultMessageNumber);
   // Pressure Line Hydraulic Filter is DIRTY
   14: XIC(inPs02PressureFilterDirty)MOVE(12,hmiFaultMessageNumber);
   // Spindle Case Line is BLOCKED
   15: XIC(inPs03MotorCaseDrain)MOVE(13,hmiFaultMessageNumber);
   // Swarf Filter is BLOCKED
   16: XIC(inPs04SwarfFilterDirty)MOVE(14,hmiFaultMessageNumber);
   // Gauge Axis Following ERROR
   17: XIC(AxisX_Gauge.FollowingError)OTL(Fault)MOVE(15,hmiFaultMessageNumber);
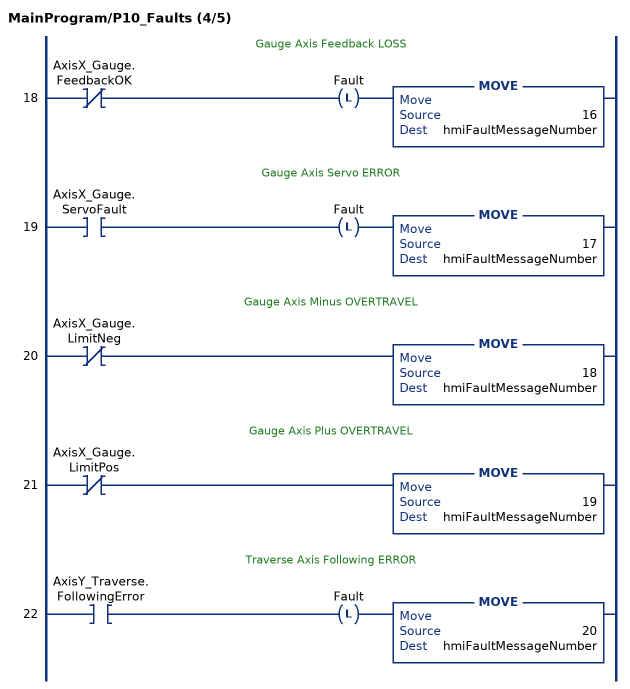
   // Gauge Axis Feedback LOSS
   18: XIO(AxisX_Gauge.FeedbackOK)OTL(Fault)MOVE(16,hmiFaultMessageNumber);
   // Gauge Axis Servo ERROR
   19: XIC(AxisX_Gauge.ServoFault)OTL(Fault)MOVE(17,hmiFaultMessageNumber);
   // Gauge Axis Minus OVERTRAVEL
   20: XIO(AxisX_Gauge.LimitNeg)MOVE(18,hmiFaultMessageNumber);
   // Gauge Axis Plus OVERTRAVEL
   21: XIO(AxisX_Gauge.LimitPos)MOVE(19,hmiFaultMessageNumber);
   // Traverse Axis Following ERROR
   22: XIC(AxisY_Traverse.FollowingError)OTL(Fault)MOVE(20,hmiFaultMessageNumber);
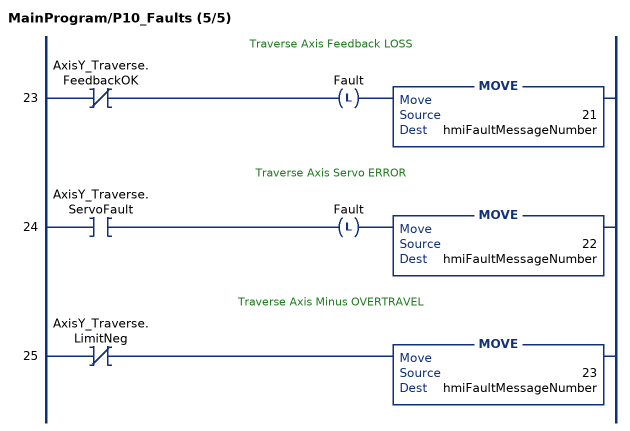
   // Traverse Axis Feedback LOSS
   23: XIO(AxisY_Traverse.FeedbackOK)OTL(Fault)MOVE(21,hmiFaultMessageNumber);
   // Traverse Axis Servo ERROR
   24: XIC(AxisY_Traverse.ServoFault)OTL(Fault)MOVE(22,hmiFaultMessageNumber);
   // Traverse Axis Minus OVERTRAVEL
   25: XIO(AxisY_Traverse.LimitNeg)MOVE(23,hmiFaultMessageNumber);
END_ROUTINE
